(*
Nazwa:			FB_SensorDiag
Opis: 			Diagnostyka czujników
Wersja:			v0.1
Data:			2024-05-27
Autor:			DP
Urzadzenia:		
Konfiguracja:	
Info:
- Diagnostyka czujnika
*)

FUNCTION_BLOCK FB_SensorDiag
VAR_INPUT
	bSensor					:BOOL;			// Wejście czujnika
	bReset					:BOOL;
	sSensorName				:STRING(200);	// Nazwa
	bShouldBlinking			:BOOL;
	tTimeToError			:TIME;			// Czas do błędu
	
	iStationIndex			:UDINT;			// Numer stacji 
	sStationName			:STRING;		// Nazwa stacji
END_VAR
VAR_OUTPUT
	bError					:BOOL;
	udiErrorID				:UDINT;	
	sErrorStationName		:STRING;							
	sErrorDescription		:STRING(200);
	sErrorDescription2		:STRING(200);	
END_VAR
VAR
	tonNoBlinkingAndOn		:TON;
	tonNoBlinkingAndOff		:TON;	
END_VAR


tonNoBlinkingAndOff	(IN:= bShouldBlinking AND NOT bSensor,	PT:=tTimeToError);
tonNoBlinkingAndOn	(IN:= bShouldBlinking AND bSensor, 		PT:=tTimeToError);
	
IF (tonNoBlinkingAndOff.Q OR tonNoBlinkingAndOn.Q) AND NOT bError THEN
	bError					:=	TRUE;
	IF tonNoBlinkingAndOff.Q THEN
		udiErrorID			:= 	1	+	iStationIndex;	
		sErrorDescription	:=	' Błąd czujnika - ciągły sygnał "0"'; 
	ELSIF tonNoBlinkingAndOn.Q THEN
		udiErrorID			:= 	2	+	iStationIndex;					
		sErrorDescription	:=	' Błąd czujnika - ciągły sygnał "1"'; 
	END_IF	
END_IF

IF bReset THEN
	bError					:=	FALSE;
END_IF

sErrorDescription2			:= sSensorName;
sErrorStationName			:= sStationName;

END_FUNCTION_BLOCK

(* stored: Version 1.1.0.1, ProductVersion 3.1.4026.13, FileIdentifier 806b344d824fd3896235d27c45633df2d0e58157, FileSignature 5984d28804ade7f6d083a7e9a68b9135180ae4a8b337ed424c23b91e95f95589f0c8113bf8ec8d3845742d7cbe9fa80cea48b79b9e864f27f9fc2e2d3d70290d955132aeef4d18a79cad3296404c5909fc51c292b918a11313483277b0edfdb9d41f7fcf3ad21f1e417550ebd7b5b47bab9d15bc4000c867c4670ac5a6adbbceba2e626bcbe1f2c586edf0bc273ee6717923b773aff38a61451b601e6763ac7039bbf2af42b365c75a142949f082b9eb40206df05739439c82742812d72b54f0fcf04a6274939dfbe7d341f1c7a84a94adb7d49f1e60ad665c49a31b0ca393ef1a836c218ab51fc0673c99ef0a67c5e920df2615039327f66d0052cccb694458
   POU FB_SensorDiag: Id {53a97ea8-1362-4349-a6ed-027b0ddb5502}, SpecialFunc None *)
